{attribute 'GeneratedUsingTerminal: EP7402-0057-0017'}
{attribute addProperty BoxType "EP7402-0057-0017"}
{attribute addProperty Id "A_0055_EP7402_0057_0018EP7402_A84790CC91"}
{attribute addProperty CRC "1192075718"}
{attribute addProperty Size "91"}
TYPE A_0054_EP7402_0057_0017_470DA1C6 EXTENDS EP7402_A84790CC :
STRUCT
	{attribute addProperty Name "A_0055_EP7402_0057_0018"}
	{attribute addProperty PreviousPort "A_0054(EP7402-0057-0017) : B"}
	A_0055_EP7402_0057_0018 : EP7402_A84790CC;
END_STRUCT
END_TYPE

(* stored: Version 1.2.0.0, ProductVersion 3.1.4024.9
   DUT A_0054_EP7402_0057_0017_470DA1C6: Id {86074087-3293-4e84-b6c5-41e30fbd75ee} *)
